INTERFACE IEnumerable EXTENDS IObject

METHOD CreateEnumerator : IEnumerator
END_METHOD

END_INTERFACE

(* stored: Version 1.1.0.1
   Itf IEnumerable: Id {dc13f336-ee79-41f7-99d1-87c5030a748a}
   Method CreateEnumerator: Id {0977fb9b-9046-4f07-b4fd-b067d11a88d4} *)
